// Implicitly generated code : DO NOT EDIT
FUNCTION CheckPointer : POINTER TO BYTE
VAR_INPUT 
	ptToTest : POINTER TO BYTE; // Destination address of the pointer
	iSize : DINT;		        // Size of the type the pointer points to. (e.g: 20 for POINTER TO ARRAY [0..9] OF INT) 
	iGran : DINT;		        // Granularity of the pointer access. This is the size of the biggest non-structured data type in the type the pointer points to. (e.g: 2 for POINTER TO ARRAY [0..9] OF INT)
	bWrite: BOOL;		        // Indicates read or write Access. TRUE = write access.
END_VAR

// No standard way of implementation. Fill your own code here
CheckPointer := ptToTest;
{flow}

END_FUNCTION

(* stored: Version 1.1.0.1, ProductVersion 3.1.4022.18
   POU CheckPointer: Id {77d871c6-61f4-4b9a-ab14-6904d1fd4b8c}, SpecialFunc CheckPointer *)
